// Mitsubishi GX Works2 project: PUMP FINAL   PLC: FX3G

PROGRAM MAIN
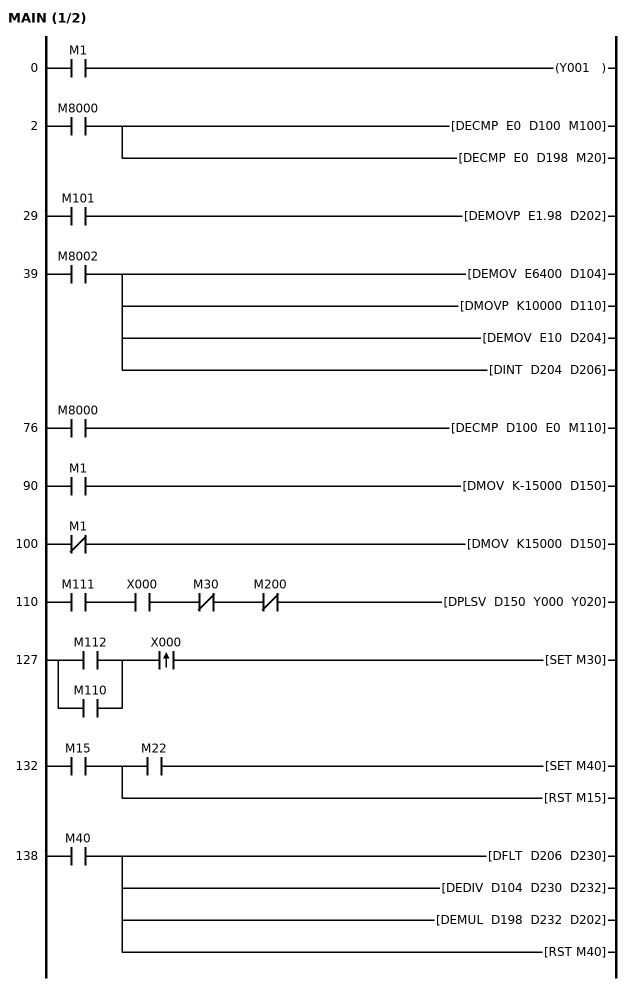
0     LD      M1
      OUT     Y001
2     LD      M8000
      DECMP   E0 D100 M100
      DECMP   E0 D198 M20
29    LD      M101
      DEMOVP  E1.98 D202
39    LD      M8002
      DEMOV   E6400 D104
      DMOVP   K10000 D110
      DEMOV   E10 D204
      DINT    D204 D206
76    LD      M8000
      DECMP   D100 E0 M110
90    LD      M1
      DMOV    K-15000 D150
100   LDI     M1
      DMOV    K15000 D150
110   LD      M111
      AND     X000
      ANI     M30
      ANI     M200
      DPLSV   D150 Y000 Y020
127   LD      M112
      OR      M110
      ANDP    X000
      SET     M30
132   LD      M15
      MPS
      AND     M22
      SET     M40
      MPP
      RST     M15
138   LD      M40
      DFLT    D206 D230
      DEDIV   D104 D230 D232
      DEMUL   D198 D232 D202
      RST     M40
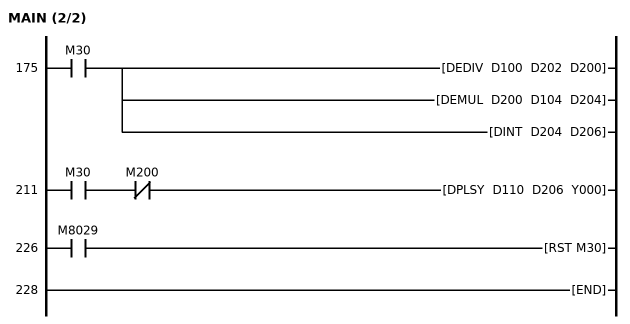
175   LD      M30
      DEDIV   D100 D202 D200
      DEMUL   D200 D104 D204
      DINT    D204 D206
211   LD      M30
      ANI     M200
      DPLSY   D110 D206 Y000
226   LD      M8029
      RST     M30
228   END
END_PROGRAM
